(* IEC 61131-3 sources: MSMP/PLC_Master/Source/Programs, 6 files *)

(* ---- PRG_Master.st ---- *)
PROGRAM PRG_Master

VAR
    Poller : FB_ModbusPolling;
    Runtime : FB_RuntimeUpdate;
END_VAR

Poller(Enable:=TRUE);
Runtime(Enable:=TRUE);

(* ---- PRG_MQTT.st ---- *)
PROGRAM PRG_MQTT
VAR
 Payload:FB_MQTTPayload;
 Json:FB_JSONBuilder;
 Gateway:FB_GatewayInterface;
END_VAR

Payload(Enable:=TRUE);
Json(Enable:=TRUE);
Gateway(Enable:=TRUE);

(* ---- PRG_Polling.st ---- *)
PROGRAM PRG_Polling
VAR
 Poll:FB_StationPolling;
 Comm:FB_CommunicationMonitor;
 Wdg:FB_MasterWatchdog;
 Counter:DWORD;
END_VAR

Poll(Enable:=TRUE);
Comm(Connected:=TRUE);
Wdg(Counter:=Counter);

(* ---- PRG_Runtime.st ---- *)
PROGRAM PRG_Runtime
VAR
 DB:FB_RuntimeDatabase;
 ST:FB_StationManager;
 AL:FB_AlarmManager;
END_VAR
DB(Enable:=TRUE);
ST(Enable:=TRUE);
AL(Enable:=TRUE);

(* ---- PRG_Scheduler.st ---- *)
PROGRAM PRG_Scheduler
VAR
 Scheduler:FB_ModbusScheduler;
 Timeout:FB_StationTimeout;
 Stats:FB_RuntimeStatistics;
END_VAR

Scheduler(Enable:=TRUE);
Timeout(CommunicationOK:=TRUE);
Stats();

(* ---- PRG_System.st ---- *)
PROGRAM PRG_System
VAR
 Payload:FB_PayloadBuilder;
 HMI:FB_HMIUpdate;
 Status:FB_SystemStatus;
END_VAR

Payload(Enable:=TRUE);
HMI(Enable:=TRUE);
Status();
